TYPE (* DataPanel Modules with low IO density DO Struct + Source Address *)
  (* Version 1.0, 2026-05-28, franz *)
  PACKAGE DataPanel::io::LO::DQ;
  IMPORT eclipse4diac::core::TypeHash;
  IMPORT DataPanel::io::LO::const::LO::LO_00;
  IMPORT DataPanel::io::LO::DQ::DataPanel_LO_DO_S;
  IMPORT DataPanel::io::LO::DQ::DataPanel_LO_DO::InvalidL;
  DataPanel_LO_DO_S_Dual_SA : STRUCT
    u8SAMember : USINT := LO_00; (* Node SA 217..224 *)
    Up : DataPanel::io::LO::DQ::DataPanel_LO_DO_S := InvalidL; (* Identify the Port 1A..4B forward, up, right, clockwise *)
    Down : DataPanel::io::LO::DQ::DataPanel_LO_DO_S := InvalidL; (* Identify the Port 1A..4B backward, down, left, counter-clockwise *)
  END_STRUCT;
END_TYPE
